TYPE CmpWorkStopMainLnSwSim :
STRUCT
	
	DBBypass: BOOL;
	ForceRFID: BOOL;
	TestRFIDData: DINT := 404;
	TestPuckData: DBGetOutputLane;

END_STRUCT
END_TYPE

(* stored: Version 1.1.0.1, ProductVersion 3.1.4024.6
   DUT CmpWorkStopMainLnSwSim: Id {228912fb-a97d-4876-840f-41c34b914705} *)
